// SIMATIC S7-200 project (STEP 7-Micro/WIN), CPU 221 REL 01.10

SYMBOL_TABLE 用户定义1
开1               I0.1
开2               I0.2
关                I0.3
关闭               I0.0
电1               Q0.1
电2               Q0.0
中点               M0.0
END_SYMBOL_TABLE

ORGANIZATION_BLOCK 主程序:OB1
TITLE=
BEGIN
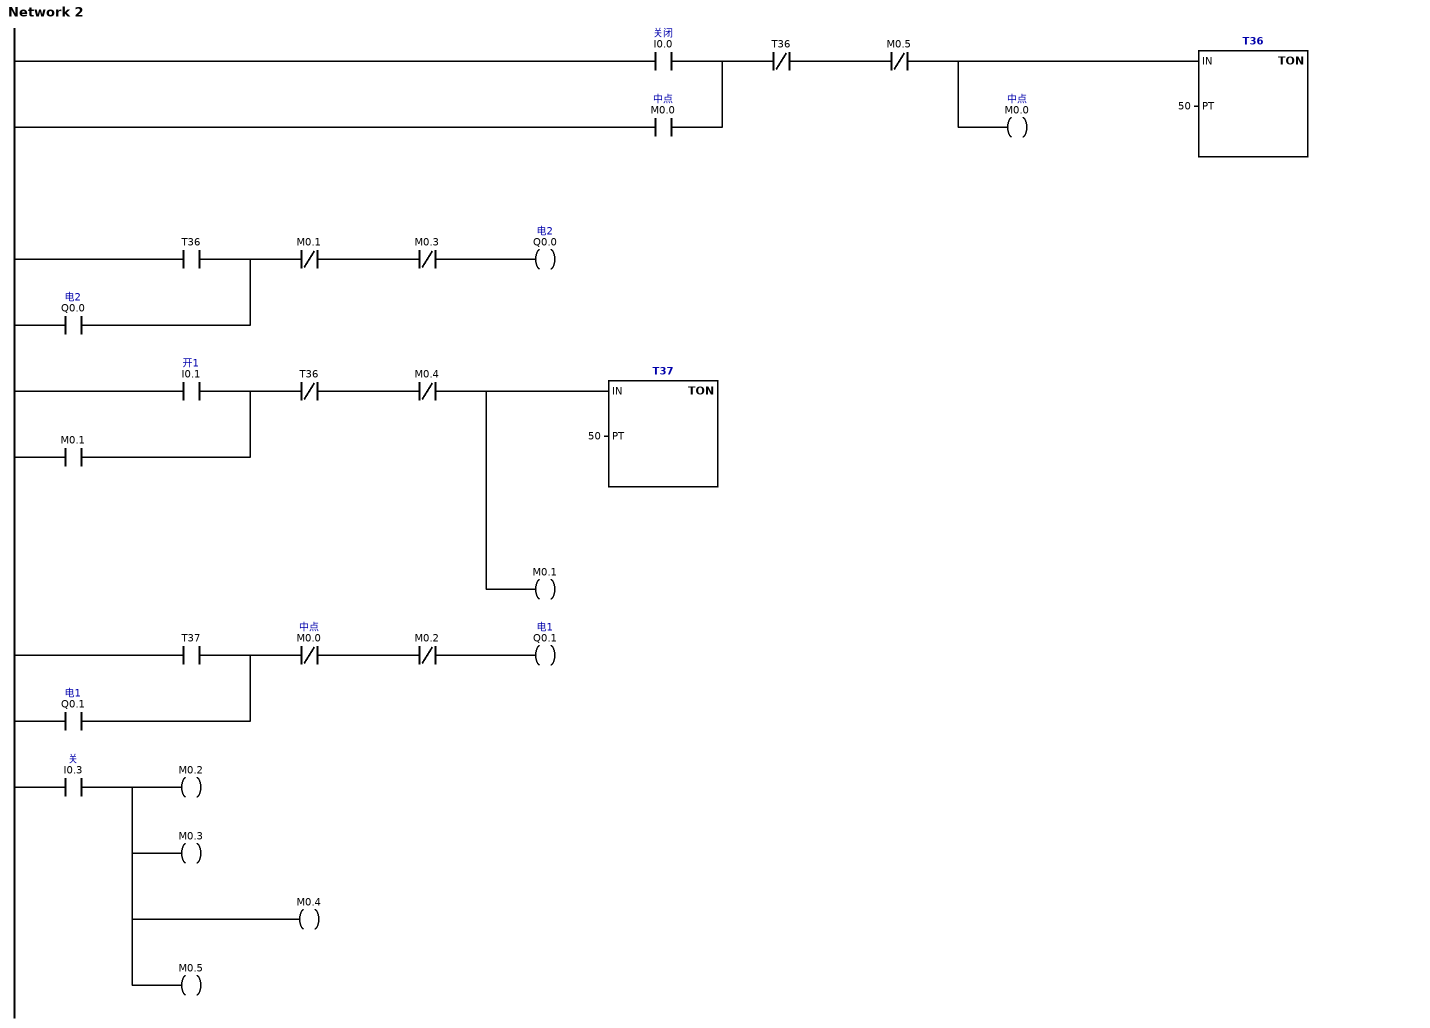
Network 2
// (network saved uncompiled; LAD cells follow)
// row 0: c0 --  c1 --  c2 --  c3 --  c4 --  c5 -| |- 关闭:I0.0 v  c6 -|/|- T36  c7 -|/|- M0.5 v  c8 --  c9 --  c10 [TON T36 IN:=power@row0, PT:=50]
// row 1: c0 --  c1 --  c2 --  c3 --  c4 --  c5 -| |- 中点:M0.0 ^  c7 ^  c8 -( ) 中点:M0.0  c10 [box]
// row 3: c0 --  c1 -| |- T36 v  c2 -|/|- M0.1  c3 -|/|- M0.3  c4 -( ) 电2:Q0.0
// row 4: c0 -| |- 电2:Q0.0  c1 -- ^
// row 5: c0 --  c1 -| |- 开1:I0.1 v  c2 -|/|- T36  c3 -|/|- M0.4 v  c4 --  c5 [TON T37 IN:=power@row5, PT:=50]
// row 6: c0 -| |- M0.1  c1 -- ^  c3 ^v  c5 [box]
// row 7: c3 ^v
// row 8: c3 ^  c4 -( ) M0.1
// row 9: c0 --  c1 -| |- T37 v  c2 -|/|- 中点:M0.0  c3 -|/|- M0.2  c4 -( ) 电1:Q0.1
// row 10: c0 -| |- 电1:Q0.1  c1 -- ^
// row 11: c0 -| |- 关:I0.3 v  c1 -( ) M0.2
// row 12: c0 ^v  c1 -( ) M0.3
// row 13: c0 ^v  c1 --  c2 -( ) M0.4
// row 14: c0 ^  c1 -( ) M0.5
END_ORGANIZATION_BLOCK
